INTERFACE I_IRC5

END_INTERFACE

(* stored: Version 1.1.0.1
   Itf I_IRC5: Id {aaf7621a-b618-424d-9754-d98352a6e316} *)
